(* IEC 61131-3 sources: CodesysTest/alpha/export/FBs/Temp Sensors/FB_TemperatureSensor.pou/TempReadingC.prop, 1 file *)

(* ---- Set.pm.st ---- *)
(*#-#-#-#-#-#-#-#-#-#---Declaration---#-#-#-#-#-#-#-#-#-#-#-#-#*)

VAR
END_VAR
(*#-#-#-#-#-#-#-#-#-#---Implementation---#-#-#-#-#-#-#-#-#-#-#-#-#*)

_temperatureReadingC := TempReadingC;
